SUBAPPLICATION Uebung_020i (* DigitalInput_I1 auf DigitalOutput_Q1; E_PULSE; Impulsformend *)
  (* Standard: 61499-2; Description: Copyright (c) 2023 Meisterschulen am Ostbahnhof This program and the accompanying materials are made available under the terms of the Eclipse Public License 2.0 which is available at https://www.eclipse.org/legal/epl-2.0/ SPDX-License-Identifier: EPL-2.0 *)
  (* Version 1.0, 2023-10-23, Franz Höpfinger, Meisterschulen am Ostbahnhof *)
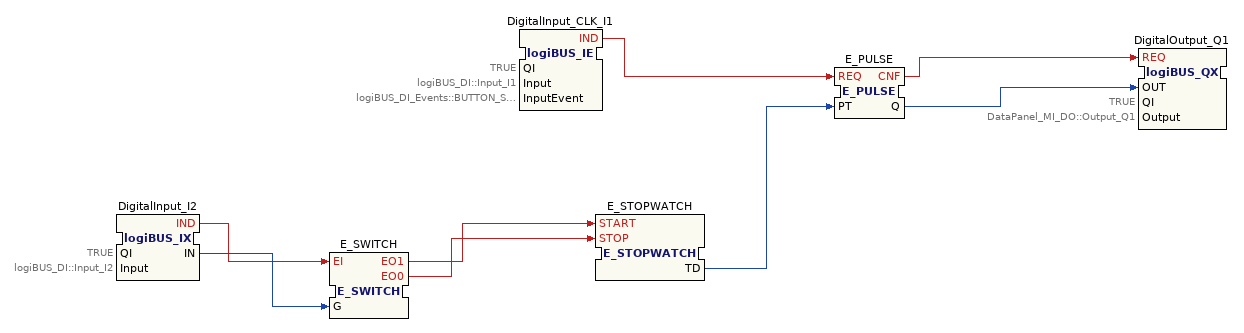
  FBS
    DigitalOutput_Q1 : logiBUS_QX(QI := TRUE, Output := DataPanel_MI_DO::Output_Q1);
    E_PULSE : E_PULSE;
    DigitalInput_CLK_I1 : logiBUS_IE(QI := TRUE, Input := logiBUS_DI::Input_I1, InputEvent := logiBUS_DI_Events::BUTTON_SINGLE_CLICK);
    E_STOPWATCH : E_STOPWATCH;
    E_SWITCH : E_SWITCH;
    DigitalInput_I2 : logiBUS_IX(QI := TRUE, Input := logiBUS_DI::Input_I2);
  END_FBS
  EVENT_CONNECTIONS
    E_PULSE.CNF TO DigitalOutput_Q1.REQ;
    DigitalInput_CLK_I1.IND TO E_PULSE.REQ;
    DigitalInput_I2.IND TO E_SWITCH.EI;
    E_SWITCH.EO1 TO E_STOPWATCH.START;
    E_SWITCH.EO0 TO E_STOPWATCH.STOP;
  END_CONNECTIONS
  DATA_CONNECTIONS
    E_PULSE.Q TO DigitalOutput_Q1.OUT;
    E_STOPWATCH.TD TO E_PULSE.PT;
    DigitalInput_I2.IN TO E_SWITCH.G;
  END_CONNECTIONS
END_SUBAPPLICATION
